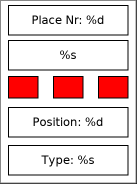
VISUALIZATION vTableFrame  // 137x184
VAR_IN_OUT
	fbTablePlace:FB_TablePlace;
	fbTableControl: FB_TableControl;
END_VAR
    Rectangle (0,0 137x184)
    Rectangle (53,76 30x22), colour toggle: fbTablePlace.stPlace.nState >=2
    Rectangle (8,76 30x22), colour toggle: fbTablePlace.stPlace.nState >=1
    Rectangle (98,76 30x22), colour toggle: fbTablePlace.stPlace.nState >=3
    Rectangle (8,5 120x30), "Place Nr: %d", text variable: fbTablePlace.stPlace.iPlaceNumber
    Rectangle (8,40 120x30), "%s", text variable: TO_STRING(fbTablePlace.stPlace.nState)
    Rectangle (8,107 120x30), "Position: %d", text variable: fbTablePlace.stPlace.iCurrentPosition
    Rectangle (98,76 30x22), invisible if: fbTablePlace.stPlace.nState<>4
    Rectangle (53,76 30x22), invisible if: fbTablePlace.stPlace.nState<>4
    Rectangle (8,76 30x22), invisible if: fbTablePlace.stPlace.nState<>4
    Rectangle (0,0 137x184)
        OnMouseDown: execute { fbTableControl.stHMI.iDialogNumber := fbTablePlace.stPlace.iPlaceNumber; }
    Rectangle (8,145 120x30), "Type: %s", text variable: TO_STRING(fbTablePlace.stPlace.nBottleType)
END_VISUALIZATION

(* stored: Version 1.1.0.1, ProductVersion 3.1.4024.15
   Visu vTableFrame: Id {27fc642f-7682-44c3-a78a-de3b0b7d87e5} *)
